// TIA Portal V15.1 export
// export: Created 2020-06-12T07:35:42.0537109Z, ExportSetting None, DisplayName Totally Integrated Automation Portal, DisplayVersion V15.1, DisplayName TIA Portal Openness, DisplayVersion V15.1, DisplayName STEP 7 Professional, DisplayVersion V15.1, DisplayName STEP 7 Safety, DisplayVersion V15.1, DisplayName WinCC Advanced, DisplayVersion V15.1
DATA_BLOCK "almai"   // DB327
{ S7_Optimized_Access := 'TRUE' }
AUTHOR : atec_osm
FAMILY : COMMON
NAME : AnaVal
VERSION : 2.0
// stored: MemoryReserve 100
   VAR
      ES1LD1_CV01 { ExternalAccessible := 'False'; ExternalVisible := 'False'; ExternalWritable := 'False'} : Bool := FALSE;   // Control Valve Dedusting System Position EN ALARM
      ES1LV1_PT01 { ExternalAccessible := 'False'; ExternalVisible := 'False'; ExternalWritable := 'False'} : Bool := FALSE;   // Vacuum Pressure MPS FL EN ALARM
      ES1LT2_XS01_volt { ExternalAccessible := 'False'; ExternalVisible := 'False'; ExternalWritable := 'False'} : Bool := FALSE;   // Actual voltage transducer EN ALARM
      ES1LT2_XS01_pwr { ExternalAccessible := 'False'; ExternalVisible := 'False'; ExternalWritable := 'False'} : Bool := FALSE;   // Actual power transducer EN ALARM
      ES1LT1_QT01 { ExternalAccessible := 'False'; ExternalVisible := 'False'; ExternalWritable := 'False'} : Bool := FALSE;   // Earth Leakage Current EN ALARM
      ES1LV1_PT02 { ExternalAccessible := 'False'; ExternalVisible := 'False'; ExternalWritable := 'False'} : Bool := FALSE;   // Air Pressure MPS RL EN ALARM
      ES1LT2_XS01_cur { ExternalAccessible := 'False'; ExternalVisible := 'False'; ExternalWritable := 'False'} : Bool := FALSE;   // Actual current transducer EN ALARM
      ES1LT1_XS01_temp1 { ExternalAccessible := 'False'; ExternalVisible := 'False'; ExternalWritable := 'False'} : Bool := FALSE;   // Transformer Actual Temperature Coil U EN ALARM
      ES1LT1_XS01_temp2 { ExternalAccessible := 'False'; ExternalVisible := 'False'; ExternalWritable := 'False'} : Bool := FALSE;   // Transformer Actual Temperature Coil V EN ALARM
      ES1LT1_XS01_temp3 { ExternalAccessible := 'False'; ExternalVisible := 'False'; ExternalWritable := 'False'} : Bool := FALSE;   // Transformer Actual Temperature Coil W EN ALARM
      ES1LA1_PT01 { ExternalAccessible := 'False'; ExternalVisible := 'False'; ExternalWritable := 'False'} : Bool := FALSE;   // Pressure Slag Bin EN ALARM
      ES1LA2_PT01 { ExternalAccessible := 'False'; ExternalVisible := 'False'; ExternalWritable := 'False'} : Bool := FALSE;   // Pressure Sluice Alloy Addion EN ALARM
      ES1LE2_M01pos { ExternalAccessible := 'False'; ExternalVisible := 'False'; ExternalWritable := 'False'} : Bool := FALSE;   // X-Adjustment Actual position EN ALARM
      ES1LE2_M02pos { ExternalAccessible := 'False'; ExternalVisible := 'False'; ExternalWritable := 'False'} : Bool := FALSE;   // Y-Adjustment Actual position EN ALARM
      ES1LC3_TT02 { ExternalAccessible := 'False'; ExternalVisible := 'False'; ExternalWritable := 'False'} : Bool := FALSE;   // Temperature Power Ram Outer Pipe RL EN ALARM
      ES1LC3_TT04 { ExternalAccessible := 'False'; ExternalVisible := 'False'; ExternalWritable := 'False'} : Bool := FALSE;   // Temperature Conduction Rail 1+2 RL EN ALARM
      ES1LC3_TT06 { ExternalAccessible := 'False'; ExternalVisible := 'False'; ExternalWritable := 'False'} : Bool := FALSE;   // Temperature Hood RL EN ALARM
      ES1LE2_XT01 { ExternalAccessible := 'False'; ExternalVisible := 'False'; ExternalWritable := 'False'} : Bool := FALSE;   // Actual Voltage Power Ram EN ALARM
      ES1LE3_PT01 { ExternalAccessible := 'False'; ExternalVisible := 'False'; ExternalWritable := 'False'} : Bool := FALSE;   // Pressure Protective Gas Hood 1 EN ALARM
      ES1LE3_PT02 { ExternalAccessible := 'False'; ExternalVisible := 'False'; ExternalWritable := 'False'} : Bool := FALSE;   // Pressure Protective Gas Hood 2 EN ALARM
      ES1LE3_QT01_O2 { ExternalAccessible := 'False'; ExternalVisible := 'False'; ExternalWritable := 'False'} : Bool := FALSE;   // Oxygen Measurement System EN ALARM
      ES1LE3_QT01_O2hw { ExternalAccessible := 'False'; ExternalVisible := 'False'; ExternalWritable := 'False'} : Bool := FALSE;   // Oxygen Measurement System EN ALARM
      ES1LE3_XT01 { ExternalAccessible := 'False'; ExternalVisible := 'False'; ExternalWritable := 'False'} : Bool := FALSE;   // Current Measuring Hood RL 1 act current EN ALARM
      ES1LE3_XT02 { ExternalAccessible := 'False'; ExternalVisible := 'False'; ExternalWritable := 'False'} : Bool := FALSE;   // Current Measuring Hood RL 2 act current EN ALARM
      ES1LE3_XT03 { ExternalAccessible := 'False'; ExternalVisible := 'False'; ExternalWritable := 'False'} : Bool := FALSE;   // Current Measuring Hood RL 3 act current EN ALARM
      ES1LE3_XT04 { ExternalAccessible := 'False'; ExternalVisible := 'False'; ExternalWritable := 'False'} : Bool := FALSE;   // Current Measuring Hood RL 4 act current EN ALARM
      ES1LZ1_PT01 { ExternalAccessible := 'False'; ExternalVisible := 'False'; ExternalWritable := 'False'} : Bool := FALSE;   // Pressure Atmosphere EN ALARM
      ES1LC1_CV01 { ExternalAccessible := 'False'; ExternalVisible := 'False'; ExternalWritable := 'False'} : Bool := FALSE;   // Actual value Control valve RL Heat Exchanger EN ALARM
      ES1LC1_PT01 { ExternalAccessible := 'False'; ExternalVisible := 'False'; ExternalWritable := 'False'} : Bool := FALSE;   // Foreward Line Strainer Pressure EN ALARM
      ES1LC1_PT02 { ExternalAccessible := 'False'; ExternalVisible := 'False'; ExternalWritable := 'False'} : Bool := FALSE;   // Return Line Strainer Pressure EN ALARM
      ES1LC1_dP02 { ExternalAccessible := 'False'; ExternalVisible := 'False'; ExternalWritable := 'False'} : Bool := FALSE;   // Differential pressure strainer EN ALARM
      ES1LC1_PT03 { ExternalAccessible := 'False'; ExternalVisible := 'False'; ExternalWritable := 'False'} : Bool := FALSE;   // Pressure CW Tank EN ALARM
      ES1LC1_QT01 { ExternalAccessible := 'False'; ExternalVisible := 'False'; ExternalWritable := 'False'} : Bool := FALSE;   // CW Tank actual conductivity EN ALARM
      ES1LC1_TT01 { ExternalAccessible := 'False'; ExternalVisible := 'False'; ExternalWritable := 'False'} : Bool := FALSE;   // CW Tank Temperature EN ALARM
      ES1LC1_TT02 { ExternalAccessible := 'False'; ExternalVisible := 'False'; ExternalWritable := 'False'} : Bool := FALSE;   // Temperature CW Recooling HE FL EN ALARM
      ES1LC1_TT03 { ExternalAccessible := 'False'; ExternalVisible := 'False'; ExternalWritable := 'False'} : Bool := FALSE;   // Temperature CW Recooling HE RL EN ALARM
      ES1LC1_TT04 { ExternalAccessible := 'False'; ExternalVisible := 'False'; ExternalWritable := 'False'} : Bool := FALSE;   // Temperature CW HE FL EN ALARM
      ES1LC3_TT01 { ExternalAccessible := 'False'; ExternalVisible := 'False'; ExternalWritable := 'False'} : Bool := FALSE;   // Temperature Electrode Column RL EN ALARM
      ES1LC5_CV01 { ExternalAccessible := 'False'; ExternalVisible := 'False'; ExternalWritable := 'False'} : Bool := FALSE;   // Control Valve CW MS1 Mould RL Position EN ALARM
      ES1LC5_CV02 { ExternalAccessible := 'False'; ExternalVisible := 'False'; ExternalWritable := 'False'} : Bool := FALSE;   // Control Valve CW MS1 Baseplate RL Position EN ALARM
      ES1LC5_FT01 { ExternalAccessible := 'False'; ExternalVisible := 'False'; ExternalWritable := 'False'} : Bool := FALSE;   // Flow CW Static Mould MS1 RL EN ALARM
      ES1LC5_FT02 { ExternalAccessible := 'False'; ExternalVisible := 'False'; ExternalWritable := 'False'} : Bool := FALSE;   // Flow CW Baseplate MS1 RL EN ALARM
      ES1LC5_PT01 { ExternalAccessible := 'False'; ExternalVisible := 'False'; ExternalWritable := 'False'} : Bool := FALSE;   // Pressure CW Melt Station 1 RL EN ALARM
      ES1LC5_PT02 { ExternalAccessible := 'False'; ExternalVisible := 'False'; ExternalWritable := 'False'} : Bool := FALSE;   // Pressure CW Baseplate 1 RL value EN ALARM
      ES1LC5_TT01 { ExternalAccessible := 'False'; ExternalVisible := 'False'; ExternalWritable := 'False'} : Bool := FALSE;   // Temperature CW Melt Station 1+2 FL EN ALARM
      ES1LC5_TT02 { ExternalAccessible := 'False'; ExternalVisible := 'False'; ExternalWritable := 'False'} : Bool := FALSE;   // Temperature CW Static Mould MS1 RL EN ALARM
      ES1LC5_TT04 { ExternalAccessible := 'False'; ExternalVisible := 'False'; ExternalWritable := 'False'} : Bool := FALSE;   // Temperature CW Baseplate 1 RL EN ALARM
      ES1LC5_TT07 { ExternalAccessible := 'False'; ExternalVisible := 'False'; ExternalWritable := 'False'} : Bool := FALSE;   // Temperature Baseplate Clamp MS1 RL EN ALARM
      ES1LC5_TT08 { ExternalAccessible := 'False'; ExternalVisible := 'False'; ExternalWritable := 'False'} : Bool := FALSE;   // Temperature Current Pipes MS1 RL EN ALARM
      ES1LC6_CV01 { ExternalAccessible := 'False'; ExternalVisible := 'False'; ExternalWritable := 'False'} : Bool := FALSE;   // Control Valve CW MS2 Mould RL Position EN ALARM
      ES1LC6_CV02 { ExternalAccessible := 'False'; ExternalVisible := 'False'; ExternalWritable := 'False'} : Bool := FALSE;   // Control Valve CW MS2 Baseplate RL Position EN ALARM
      ES1LC6_FT01 { ExternalAccessible := 'False'; ExternalVisible := 'False'; ExternalWritable := 'False'} : Bool := FALSE;   // Flow CW Static Mould MS2 RL EN ALARM
      ES1LC6_FT02 { ExternalAccessible := 'False'; ExternalVisible := 'False'; ExternalWritable := 'False'} : Bool := FALSE;   // Flow CW Baseplate 2 RL EN ALARM
      ES1LC6_PT01 { ExternalAccessible := 'False'; ExternalVisible := 'False'; ExternalWritable := 'False'} : Bool := FALSE;   // Pressure CW Melt Station 2 RL EN ALARM
      ES1LC6_PT02 { ExternalAccessible := 'False'; ExternalVisible := 'False'; ExternalWritable := 'False'} : Bool := FALSE;   // Pressure CW Baseplate 2 RL value EN ALARM
      ES1LC6_TT02 { ExternalAccessible := 'False'; ExternalVisible := 'False'; ExternalWritable := 'False'} : Bool := FALSE;   // Temperature CW Static Mould MS2 RL EN ALARM
      ES1LC6_TT04 { ExternalAccessible := 'False'; ExternalVisible := 'False'; ExternalWritable := 'False'} : Bool := FALSE;   // Temperature CW Baseplate 2 RL EN ALARM
      ES1LC6_TT07 { ExternalAccessible := 'False'; ExternalVisible := 'False'; ExternalWritable := 'False'} : Bool := FALSE;   // Temperature Baseplate Clamp MS2 RL Actual value
      ES1LC6_TT08 { ExternalAccessible := 'False'; ExternalVisible := 'False'; ExternalWritable := 'False'} : Bool := FALSE;   // Temperature Current Pipes MS2 RL EN ALARM
      ES1LC7_CV01 { ExternalAccessible := 'False'; ExternalVisible := 'False'; ExternalWritable := 'False'} : Bool := FALSE;   // Control Valve CW Module Recooling HE RL Position EN ALARM
      ES1LC7_PT10 { ExternalAccessible := 'False'; ExternalVisible := 'False'; ExternalWritable := 'False'} : Bool := FALSE;   // Pressure CW Module Pump FL EN ALARM
      ES1LC7_TT01 { ExternalAccessible := 'False'; ExternalVisible := 'False'; ExternalWritable := 'False'} : Bool := FALSE;   // Temperature CW Transductor RL EN ALARM
      ES1LC7_TT02 { ExternalAccessible := 'False'; ExternalVisible := 'False'; ExternalWritable := 'False'} : Bool := FALSE;   // Temperature CW Current Condution F&amp;B RL EN ALARM
      ES1LC7_TT10 { ExternalAccessible := 'False'; ExternalVisible := 'False'; ExternalWritable := 'False'} : Bool := FALSE;   // Temperature CW Module Pump FL EN ALARM
      ES1LC7_TT12 { ExternalAccessible := 'False'; ExternalVisible := 'False'; ExternalWritable := 'False'} : Bool := FALSE;   // Temperature CW Module HE FL EN ALARM
      ES1LC7_TT13 { ExternalAccessible := 'False'; ExternalVisible := 'False'; ExternalWritable := 'False'} : Bool := FALSE;   // Temperature CW Module HE RL EN ALARM
      ES1LC7_TT14 { ExternalAccessible := 'False'; ExternalVisible := 'False'; ExternalWritable := 'False'} : Bool := FALSE;   // Temperature CW Module Recooling HE RL EN ALARM
      ES1LC7_TT15 { ExternalAccessible := 'False'; ExternalVisible := 'False'; ExternalWritable := 'False'} : Bool := FALSE;   // Temperature CW Module Recooling HE FL EN ALARM
      ES1LC7_TT16 { ExternalAccessible := 'False'; ExternalVisible := 'False'; ExternalWritable := 'False'} : Bool := FALSE;   // Temperature CW Vacuum Dry Screw Pump RL EN ALARM
      ES1LC7_TT17 { ExternalAccessible := 'False'; ExternalVisible := 'False'; ExternalWritable := 'False'} : Bool := FALSE;   // Temperature CW Vacuum Roots Pump RL EN ALARM
      ES1LG1_CV01 { ExternalAccessible := 'False'; ExternalVisible := 'False'; ExternalWritable := 'False'} : Bool := FALSE;   // Control Valve Ar PGH Act Flow EN ALARM
      ES1LG1_CV02 { ExternalAccessible := 'False'; ExternalVisible := 'False'; ExternalWritable := 'False'} : Bool := FALSE;   // Control Valve N2 PGH Act Flow EN ALARM
      ES1LA1_WT01 { ExternalAccessible := 'False'; ExternalVisible := 'False'; ExternalWritable := 'False'} : Bool := FALSE;   // Weight Slag Bin EN ALARM
      ES1LA2_WT01 { ExternalAccessible := 'False'; ExternalVisible := 'False'; ExternalWritable := 'False'} : Bool := FALSE;   // Weight Alloy Bin EN ALARM
      ES1LE1_WT01 { ExternalAccessible := 'False'; ExternalVisible := 'False'; ExternalWritable := 'False'} : Bool := FALSE;   // Weight Electrode Weight EN ALARM
   END_VAR
BEGIN
END_DATA_BLOCK
